PROGRAM P_ControlBlock
VAR
	fbDeadBandTester : FB_DeadbandTester;
	fbAutoClock : FB_AutoClock;
	fbMotionRef : FB_MotionRef;
	fbControl : FB_ControlSignal;
	fbInitialPos : FB_InitialPos;
END_VAR


fbInitialPos(
	bEnable := G_Mode.bRunning,
	fCurrentPos := G_OPC.fPistonPosition
);

fbMotionRef(
	fInitialPos := fbInitialPos.fInitialPos
);

IF G_Mode.bAuto AND G_Mode.bRunning THEN

//fbInitialPos(
//	bEnable := G_Inputs.bStartButton,
//	fCurrentPos := G_OPC.fPistonPosition
//);

fbAutoClock(
	fStart := G_Inputs.bStartButton,
	fRunning := G_Mode.bRunning,
	fCycle := G_Parameter.fCycleTime
);

fbMotionRef(
	fTime := fbAutoClock.fTime,
	fAmplitude := G_Parameter.fAmplitude,
	//fInitialPos := fbInitialPos.fInitialPos,
	fFrequency := G_Parameter.fFrequency,
	fXDotRef => G_OPC.fXDotRef,
	fXRef => G_OPC.fXRef 
);

fbControl(
	fUFF := G_OPC.fUFF,
	fPID := G_OPC.fSignalPID,
	bEnableU := G_Enables.bEnableU,
	fQMaxUp := G_Parameter.fQMaxUp,
	fQMaxDown := G_Parameter.fQMaxDown,
	fDeadUp := G_Parameter.fDeadUp,
	fDeadDown := G_Parameter.fDeadDown,
	fXDotRef := G_OPC.fXDotRef,
	fError := G_OPC.fError,
	
	fU => G_OPC.fU
);

ELSIF G_Mode.bManual AND G_Mode.bRunning THEN

//fbInitialPos(
//	bEnable := G_Inputs.bStartButton,
//	fCurrentPos := G_OPC.fPistonPosition
//);

fbDeadBandTester(
	fInput := G_OPC.fJoystick,
	bEnable := G_Enables.bDeadBandTest,
	fConst := G_Parameter.fConst,
	fOutput => G_OPC.fU
);

END_IF

END_PROGRAM

(* stored: Version 1.1.0.1, ProductVersion 3.1.4024.12
   POU P_ControlBlock: Id {34b73f17-fb3f-4014-8571-592d49402d29}, SpecialFunc None *)
